Staubli VAL3: writeFloatValue.pgx

public program writeFloatValue(num x_nCamID (dimensions=1), string x_sCellNumber (dimensions=1), num x_nValue (dimensions=1), bool& x_bError[] (dimensions=1))
  local string l_sCell
  local bool l_bIsOk
begin
  //-----------------------------------------------------------------------
  //Header begin
  //Description of program
  //  Sets an edit box control contained in a cell (x_sCellNumber)
  //  to a specified floating-point value (x_nValue)
  //  The target cell of the writing operation in the Cognex spreadsheet must
  //  be of the EditFloat type.
  //
  //Input parameters
  //  num x_nCamID :
  //    role : camera's ID
  //  string x_sCellNumber :
  //    role : The column letter and the row number of the cell value to get.
  //    possible values : - column letter : (A to Z)
  //                      - row number : (000 to 399)
  //  num x_nValue :
  //    role : value to writing in the cell
  //
  //Output parameters
  //  bool x_bError :
  //    role : returns true if an error occurred and false otherwise
  //
  //Examples
  //  call writeFloatValue(nCamID,"C6",5.6,l_bError)
  //
  //History
  //  Creation : 19-05-08 - f.Rob
  //Header end
  //-----------------------------------------------------------------------

  // Write a float value into a cell
  x_bError=true
  call checkCellFormat(x_nCamID,x_sCellNumber,l_bIsOk)
  if l_bIsOk
    nProgram[x_nCamID]=9
    call sendCommand(x_nCamID,"SF"+x_sCellNumber+toString("0.5",x_nValue),x_bError)
  endIf
end
